{attribute 'GeneratedUsingTerminal: EKM1101-0000-0016'}
{attribute addProperty BoxType "EKM1101-0000-0016"}
{attribute addProperty Description "EKM1101 EtherCAT Coupler  (2A E-Bus, ID switch, Diagnostics, isolated)"}
{attribute addProperty Physics "YKY"}
{attribute addProperty Id "MMS_Device_InputsAT %I*MMS_Device_Inputs_ADC3123E5MMS_Acceleration_StatusAT %I*MMS_Acceleration_Status_117690999MMS_Acceleration_X_AxisAT %I*MMS_Acceleration_X_Axis_80E77D6A2MMS_Acceleration_Y_AxisAT %I*MMS_Acceleration_Y_Axis_80E77D6A2MMS_Acceleration_Z_AxisAT %I*MMS_Acceleration_Z_Axis_80E77D6A2MMS_Acceleration_TimestampAT %I*MMS_Acceleration_Timestamp_8B9FE1A28MMS_Voltage_Us_In_InputsAT %I*MMS_Voltage_Us_In_Inputs_60D55C7211MMS_Voltage_Up_In_InputsAT %I*MMS_Voltage_Up_In_Inputs_60D55C7211MMS_Voltage_Up_Out_InputsAT %I*MMS_Voltage_Up_Out_Inputs_60D55C7211MMS_Device_OutputsAT %Q*MMS_Device_Outputs_E6E6F9D11WcStateAT %I*WcState_9091E0EB2InfoDataAT %I*InfoData_BEF6B88E18"}
{attribute addProperty CRC "2134996514"}
{attribute addProperty Size "82"}
TYPE EKM1101_7F417622 EXTENDS EtcSlaveBoxBase_77A0E4A7 :
STRUCT
	{attribute addProperty Name "MMS_Device_Inputs"}
	MMS_Device_Inputs : MMS_Device_Inputs_ADC3123E;
	{attribute addProperty Name "MMS_Acceleration_Status"}
	MMS_Acceleration_Status : MMS_Acceleration_Status_11769099;
	{attribute addProperty Name "MMS_Acceleration_X_Axis"}
	MMS_Acceleration_X_Axis : MMS_Acceleration_X_Axis_80E77D6A;
	{attribute addProperty Name "MMS_Acceleration_Y_Axis"}
	MMS_Acceleration_Y_Axis : MMS_Acceleration_Y_Axis_80E77D6A;
	{attribute addProperty Name "MMS_Acceleration_Z_Axis"}
	MMS_Acceleration_Z_Axis : MMS_Acceleration_Z_Axis_80E77D6A;
	{attribute addProperty Name "MMS_Acceleration_Timestamp"}
	MMS_Acceleration_Timestamp : MMS_Acceleration_Timestamp_8B9FE1A2;
	{attribute addProperty Name "MMS_Voltage_Us_In_Inputs"}
	MMS_Voltage_Us_In_Inputs : MMS_Voltage_Us_In_Inputs_60D55C72;
	{attribute addProperty Name "MMS_Voltage_Up_In_Inputs"}
	MMS_Voltage_Up_In_Inputs : MMS_Voltage_Up_In_Inputs_60D55C72;
	{attribute addProperty Name "MMS_Voltage_Up_Out_Inputs"}
	MMS_Voltage_Up_Out_Inputs : MMS_Voltage_Up_Out_Inputs_60D55C72;
	{attribute addProperty Name "MMS_Device_Outputs"}
	MMS_Device_Outputs : MMS_Device_Outputs_E6E6F9D1;
	{attribute addProperty Name "WcState"}
	WcState : WcState_9091E0EB;
	{attribute addProperty Name "InfoData"}
	InfoData : InfoData_BEF6B88E;
END_STRUCT
END_TYPE

(* stored: Version 1.2.0.0, ProductVersion 3.1.4024.9
   DUT EKM1101_7F417622: Id {f6afb99a-adb6-48c1-80dd-260cb1a1c88f} *)
